// TIA Portal V21 export
DATA_BLOCK "TemperatureControl"   // DB303
AUTHOR : PRECISE
FAMILY : PRECISE
// stored: AutoNumber false, InstanceOfName FB311, InstanceOfType FB
"FB311"
   // VAR_INPUT
   //    Enable : Bool;
   //    Disable : Bool;
   //    Fault : Bool;
   //    SecPulse : Bool;
   //    AlwaysTrue : Bool;
   //    StartConfirmationPopupSel : Bool;
   //    EndConfirmationPopupSel : Bool;
   //    TimebaseSel : Bool;
   //    TemperatureMaintainSel : Bool;
   //    BypassSel : Bool := true;
   //    JacketAirPurgingSel : Bool;
   //    TemperatureControlSel : Int;
   //    SensorSel : Int;
   //    BatchSizeSel : Int;
   //    HeatingUtilitySel : Int;
   //    CoolingUtilitySelection : Int := 0;
   //    SetTemperature : Real;
   //    TimeMin : Int := 1;
   //    TimeSec : Int := 30;
   //    ActualTemperatureVessel : Real;
   //    ActualTemperatureJacket : Real;
   //    JVDelay : Int;
   //    JDDelay : Int;
   //    TemperatureTol : Real;
   //    CoolingThreshold : Real;
   //    ChillingThreshold : Real;
   //    HeatHighTemperatureTol : Real;
   //    CoolLowTemperatureTol : Real;
   //    JacketAirPurgingTimeSec : Int;
   // END_VAR
   // VAR_OUTPUT
   //    JacketAirValve : Bool;
   //    BypassValve : Bool;
   //    JacketVentValve1 : Bool;
   //    JacketDrainValve1 : Bool;
   //    CoolingWaterInletValve1 : Bool;
   //    CoolingWaterOutletValve1 : Bool;
   //    ChilledWaterInletValve1 : Bool;
   //    ChilledWaterOutletValve1 : Bool;
   //    BrineWaterInletValve1 : Bool;
   //    BrineWaterOutletValve1 : Bool;
   //    HotWaterInletValve1 : Bool;
   //    HotWaterOutletValve1 : Bool;
   //    SteamInlet1 : Bool;
   //    Condensateoutlet1 : Bool;
   //    JacketVentValve2 : Bool;
   //    JacketDrainValve2 : Bool;
   //    CoolingWaterInletValve2 : Bool;
   //    CoolingWaterOutletValve2 : Bool;
   //    ChilledWaterInletValve2 : Bool;
   //    ChilledWaterOutletValve2 : Bool;
   //    BrineWaterInletValve2 : Bool;
   //    BrineWaterOutletValve2 : Bool;
   //    HotWaterInletValve2 : Bool;
   //    HotWaterOutletValve2 : Bool;
   //    SteamInlet2 : Bool;
   //    Condensateoutlet2 : Bool;
   //    AlarmHeatHighTemperature : Bool;
   //    AlarmCoolLowTemperature : Bool;
   //    StartConfirmationPopup : Bool;
   //    EndConfirmationPopup : Bool;
   //    JacketAirPurgingPopup : Bool;
   //    TimeMinPV : DInt;
   //    TimeSecPV : DInt;
   //    JacketAirPurgingTimeSecPV : Int;
   //    PrintTrigger : Bool;
   //    PrintWord : Int;
   //    PrintStatus : String[50];
   // END_VAR
   // VAR_IN_OUT
   //    Start : Bool;
   //    Stop : Bool;
   //    Reset : Bool;
   //    StartConfirmationAck : Bool;
   //    EndConfirmationAck : Bool;
   //    JacketAirPurgingAck : Bool;
   //    AlarmAck : Bool;
   //    SpareBtn1 : Bool;
   //    Running : Bool;
   //    Selected : Bool;
   //    Paused : Bool;
   //    StartConfirmationPopupTemp : Bool;
   //    EndConfirmationPopupTemp : Bool;
   //    Started : Bool;
   //    Over : Bool;
   //    StartJVDelay : Bool := 1;
   //    StartJDDelay : Bool;
   //    StartUtility : Bool;
   //    StartChilling : Bool;
   //    StartBrine : Bool;
   //    StartJacketAirPurging : Bool;
   //    HeatTempReached : Bool;
   //    CoolTempReached : Bool;
   //    TemperatureTolNeg : Real;
   //    TemperatureTolPos : Real;
   //    HeatHighTemperatureTolCal : Real;
   //    CoolLowTemperatureTolCal : Real;
   //    JacketPressureSelection : Bool;
   //    JacketPressureReached : Bool;
   //    JacketUtilityPressureValve : Bool;
   //    JAcketAlarms : Bool;
   //    Temp : Bool;
   //    JacketTime : Int;
   //    JacketSafetyPressure : Real;
   //    JAcketActPressure : Real;
   // END_VAR
   // VAR
   //    PrintTriggerTemp : Bool;
   //    RE1 : Bool;
   //    RE2 : Bool;
   //    RE3 : Bool;
   //    RE4 : Bool;
   //    RE5 : Bool;
   //    RE6 : Bool;
   //    RE7 : Bool;
   //    RE8 : Bool;
   //    RE9 : Bool;
   //    RE10 : Bool;
   //    RE11 : Bool;
   //    "Timer" : "FB101";
   //    PrintTriggerResetTimer { S7_SetPoint := 'True'} : TON_TIME;
   //    BtnResetTimer { S7_SetPoint := 'True'} : TON_TIME;
   //    JVDelayTime { S7_SetPoint := 'True'} : "FB103";
   //    JDDelayTime { S7_SetPoint := 'True'} : "FB103";
   //    JAPTime { S7_SetPoint := 'True'} : "FB103";
   //    ActualTemperature : Real;
   //    JacketpressureTimer { S7_SetPoint := 'True'} : "FB103";
   //    FB101_Instance { S7_SetPoint := 'True'} : "FB101";
   // END_VAR
BEGIN
END_DATA_BLOCK
